FUNCTION_BLOCK RegisterServiceOpcUaOriginal (* Register Service using OPC UA *)
  (* Standard: 61499-2; Description: Copyright (c) 2019 fortiss GmbH This program and the accompanying materials are made available under the terms of the Eclipse Public License 2.0 which is available at https://www.eclipse.org/legal/epl-2.0/ SPDX-License-Identifier: EPL-2.0 *)
  (* Version 1.0, 2019-09-17, Jose Cabral, fortiss GmbH *)
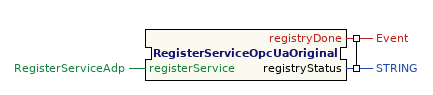
  EVENT_OUTPUT
    registryDone WITH registryStatus;
  END_EVENT
  VAR_OUTPUT
    registryStatus : STRING;
  END_VAR
  SOCKETS
    registerService : RegisterServiceAdp; (* Register Service adapter *)
  END_SOCKETS
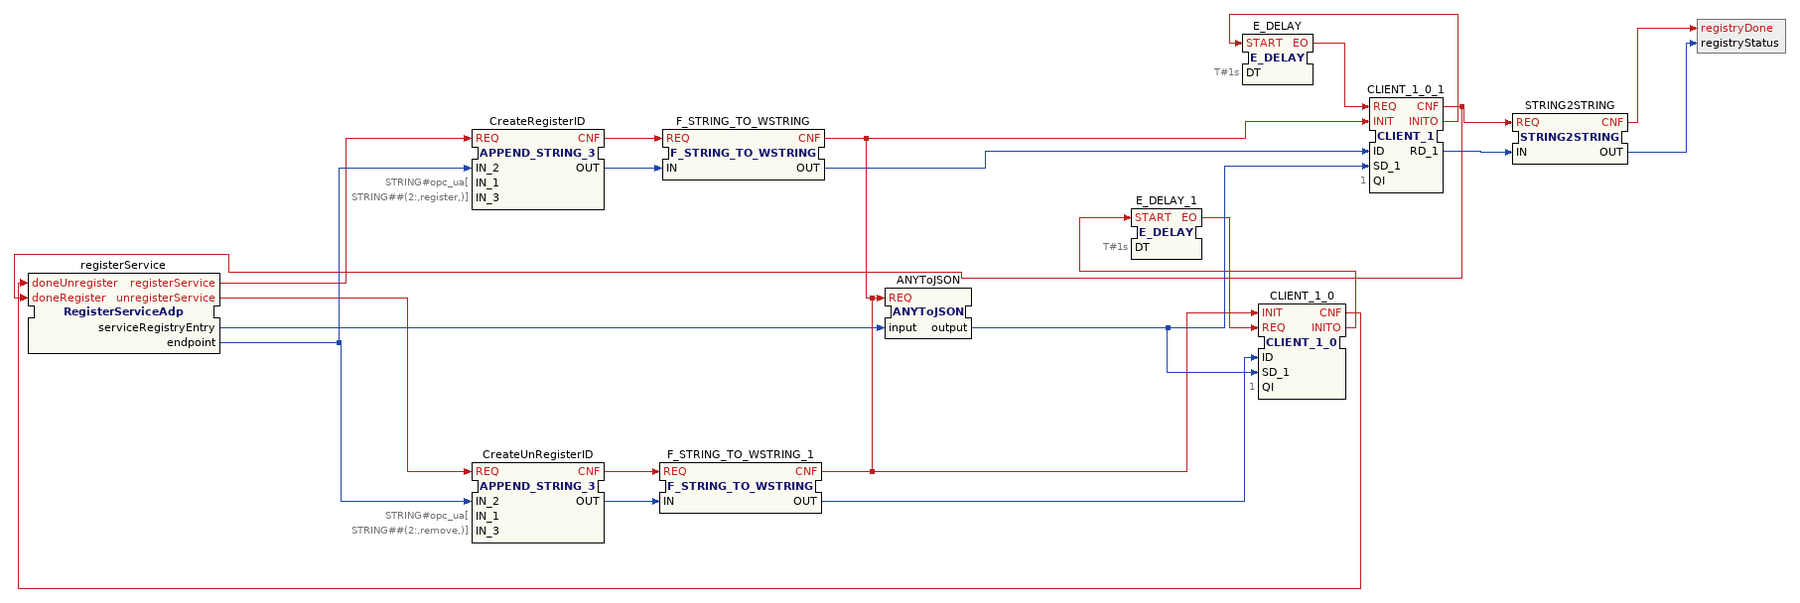
  FBS
    CreateRegisterID : APPEND_STRING_3(IN_1 := STRING#opc_ua[, IN_3 := STRING##(2:,register,)]);
    F_STRING_TO_WSTRING : F_STRING_TO_WSTRING;
    CreateUnRegisterID : APPEND_STRING_3(IN_1 := STRING#opc_ua[, IN_3 := STRING##(2:,remove,)]);
    F_STRING_TO_WSTRING_1 : F_STRING_TO_WSTRING;
    ANYToJSON : ANYToJSON;
    CLIENT_1_0 : CLIENT_1_0(QI := 1);
    CLIENT_1_0_1 : CLIENT_1(QI := 1);
    STRING2STRING : STRING2STRING;
    E_DELAY : E_DELAY(DT := T#1s);
    E_DELAY_1 : E_DELAY(DT := T#1s);
  END_FBS
  EVENT_CONNECTIONS
    CreateRegisterID.CNF TO F_STRING_TO_WSTRING.REQ;
    CreateUnRegisterID.CNF TO F_STRING_TO_WSTRING_1.REQ;
    F_STRING_TO_WSTRING.CNF TO ANYToJSON.REQ;
    F_STRING_TO_WSTRING_1.CNF TO ANYToJSON.REQ;
    registerService.registerService TO CreateRegisterID.REQ;
    registerService.unregisterService TO CreateUnRegisterID.REQ;
    CLIENT_1_0.CNF TO registerService.doneUnregister;
    CLIENT_1_0_1.CNF TO registerService.doneRegister;
    CLIENT_1_0_1.CNF TO STRING2STRING.REQ;
    STRING2STRING.CNF TO registryDone;
    E_DELAY.EO TO CLIENT_1_0_1.REQ;
    CLIENT_1_0_1.INITO TO E_DELAY.START;
    F_STRING_TO_WSTRING.CNF TO CLIENT_1_0_1.INIT;
    F_STRING_TO_WSTRING_1.CNF TO CLIENT_1_0.INIT;
    CLIENT_1_0.INITO TO E_DELAY_1.START;
    E_DELAY_1.EO TO CLIENT_1_0.REQ;
  END_CONNECTIONS
  DATA_CONNECTIONS
    CreateRegisterID.OUT TO F_STRING_TO_WSTRING.IN;
    CreateUnRegisterID.OUT TO F_STRING_TO_WSTRING_1.IN;
    registerService.serviceRegistryEntry TO ANYToJSON.input;
    registerService.endpoint TO CreateRegisterID.IN_2;
    registerService.endpoint TO CreateUnRegisterID.IN_2;
    F_STRING_TO_WSTRING.OUT TO CLIENT_1_0_1.ID;
    ANYToJSON.output TO CLIENT_1_0_1.SD_1;
    CLIENT_1_0_1.RD_1 TO STRING2STRING.IN;
    STRING2STRING.OUT TO registryStatus;
    F_STRING_TO_WSTRING_1.OUT TO CLIENT_1_0.ID;
    ANYToJSON.output TO CLIENT_1_0.SD_1;
  END_CONNECTIONS
END_FUNCTION_BLOCK
